PROGRAM MAIN
VAR
END_VAR

END_PROGRAM

(* stored: Version 1.1.0.1
   POU MAIN: Id {4045dbca-0452-4086-99a5-68925e31f21f} *)
